Universal Robots URScript: box_placing_pr1.script

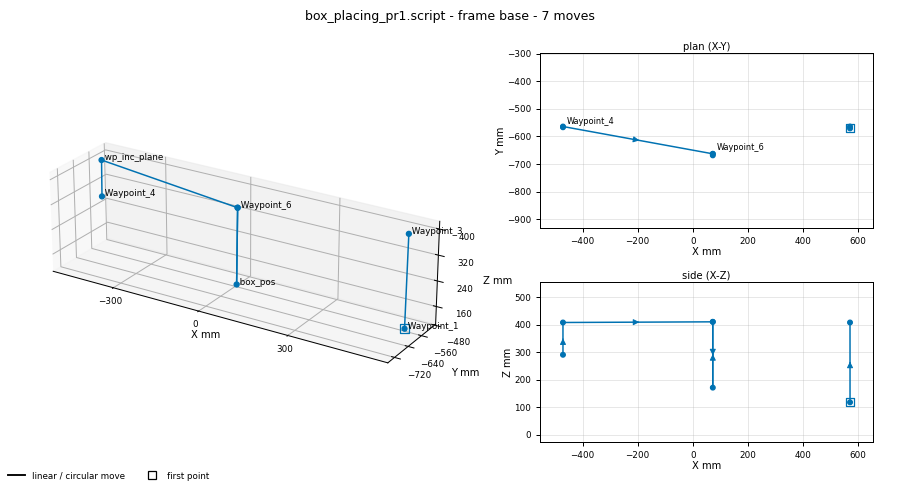
[picture p0: tool path of box_placing_pr1.script in frame base, 7 of 8 moves have a stored position in this frame; points joined in program order, loops and branches not executed]
def box_placing_pr1():
  set_safety_mode_transition_hardness(1)
  set_tcp(p[0.0,0.0,0.0,0.0,0.0,0.0])
  set_payload(0.0)
  set_gravity([0.0, 0.0, 9.82])
  set_standard_analog_input_domain(0, 1)
  set_standard_analog_input_domain(1, 1)
  set_tool_analog_input_domain(0, 1)
  set_tool_analog_input_domain(1, 1)
  set_analog_outputdomain(0, 0)
  set_analog_outputdomain(1, 0)
  set_tool_voltage(24)
  set_input_actions_to_default()
  set_tool_communication(False, 115200, 0, 1, 1.5, 3.5)
  set_tool_output_mode(0)
  set_tool_digital_output_mode(0, 3)
  set_tool_digital_output_mode(1, 3)
  global box_placing_1=p[0.5729530147544537,-0.5700957532331434,0.10756608120479487,5.789473277800655E-5,-0.0372445138718035,-3.14136724439086]
  global pox_place=p[-0.48281559147672787,-0.5676153780257446,0.24858418286268774,0.0744679787965601,2.6697818535523212,-0.722806939486385]
  global Waypoint_1_p=p[.571350906774, -.570754339342, .117565005607, -.000021746886, 3.140014852606, -.000050447991]
  global Waypoint_1_q=[2.1442551612854004, -0.9957612317851563, 1.9401515165912073, -2.517834325829977, -1.5707781950580042, 0.5653424263000488]
  global Waypoint_3_p=p[.571257104046, -.563837393624, .407498540114, -.000151158778, 3.140007692731, -.000026398933]
  global Waypoint_3_q=[2.149075984954834, -1.3216117185405274, 1.7802642027484339, -2.0321041546263636, -1.5740817228900355, 0.5716409683227539]
  global Waypoint_2_from_p=p[-.482827972204, -.567597285845, .248569345138, .074551946327, 2.669726244445, -.722810613786]
  global Waypoint_2_to_p=p[-.482797082425, -.563859017260, .407490097055, .074459411645, 2.669770137388, -.722783710165]
  global Waypoint_4_p=p[-.471150063525, -.566651664562, .290163680256, -.000107423198, 3.140028197571, -.000018987743]
  global Waypoint_4_q=[0.6442923545837561, -1.3084982198527868, 2.008158032094214, -2.270989080468979, -1.5736134688007617, -0.9346278349506782]
  global wp_inc_plane_p=p[-.471170481321, -.563844358818, .407460144481, -.000023857309, 3.139999358685, .000022690335]
  global wp_inc_plane_q=[0.6411652565002441, -1.4266775411418458, 1.9097407499896448, -2.0543533764281214, -1.5749347845660608, -0.9366801420794886]
  global Waypoint_6_p=p[.072941651956, -.662968779906, .409842477860, -.000047182021, 3.140039073033, -.000023180941]
  global Waypoint_6_q=[1.4225287437438965, -1.5383246702006836, 2.029053036366598, -2.06308712581777, -1.5748990217791956, -0.1556795279132288]
  global box_pos_p=p[.072975237359, -.668625191092, .170861527187, -.000069484777, 3.139978897906, -.000033254883]
  global box_pos_q=[1.4236183166503906, -1.2257078450969239, 2.197754208241598, -2.544392248193258, -1.571258846913473, -0.1564572493182581]
  global Waypoint_5_p=p[.072932217313, -.662956319476, .409868936128, .000008626569, 3.140004745684, -.000050597097]
  global Waypoint_5_q=[1.4225049018859863, -1.538372353916504, 2.029053036366598, -2.0630513630309046, -1.5748627821551722, -0.15566760698427373]
  while (True):
    $ 1 "Robot Program"
    $ 2 "MoveL"
    $ 3 "Waypoint_1"
    movel(pose_trans(box_placing_1, pose_trans(p[.572954085294, -.572488182458, -.093998318537, -.000057894727, .037244513871, 3.141367244343], Waypoint_1_p)), a=1.2, v=0.1)
    $ 4 "Waypoint_3"
    movel(pose_trans(box_placing_1, pose_trans(p[.572954085294, -.572488182458, -.093998318537, -.000057894727, .037244513871, 3.141367244343], Waypoint_3_p)), a=1.2, v=0.1, r=0.05)
    $ 5 "Waypoint_2"
    movel(pose_add(get_target_tcp_pose(), pose_sub(Waypoint_2_to_p, Waypoint_2_from_p)), a=1.2, v=0.1)
    $ 6 "Waypoint_4"
    movel(pose_trans(box_placing_1, pose_trans(p[.572954085294, -.572488182458, -.093998318537, -.000057894727, .037244513871, 3.141367244343], Waypoint_4_p)), a=1.2, v=0.1)
    $ 7 "wp_inc_plane"
    movel(pose_trans(box_placing_1, pose_trans(p[.572954085294, -.572488182458, -.093998318537, -.000057894727, .037244513871, 3.141367244343], wp_inc_plane_p)), a=1.2, v=0.1)
    $ 8 "Waypoint_6"
    movel(pose_trans(box_placing_1, pose_trans(p[.572954085294, -.572488182458, -.093998318537, -.000057894727, .037244513871, 3.141367244343], Waypoint_6_p)), a=1.2, v=0.1)
    $ 9 "box_pos"
    movel(pose_trans(box_placing_1, pose_trans(p[.572954085294, -.572488182458, -.093998318537, -.000057894727, .037244513871, 3.141367244343], box_pos_p)), a=1.2, v=0.1)
    $ 10 "Waypoint_5"
    movel(pose_trans(box_placing_1, pose_trans(p[.572954085294, -.572488182458, -.093998318537, -.000057894727, .037244513871, 3.141367244343], Waypoint_5_p)), a=1.2, v=0.1)
  end
end
